FUNCTION f_MessageSet : BOOL
VAR_INPUT
  stMessage   : ST_Message;
END_VAR
VAR
  uiIndex   : INT;
  uiFound   : INT;
END_VAR

stMessage.tTime := GVL_AXIS_CTRL.gsLocalTime;

FOR uiIndex := 1 TO GVL_AXIS_CTRL.gciMaxMessage
DO
  IF (GVL_AXIS_CTRL.gatMessages[uiIndex].eType = e_MessageType.eMessageEmpty)
  THEN
    GVL_AXIS_CTRL.gatMessages[uiIndex] := stMessage;
    GVL_AXIS_CTRL.giMsgIndex := uiIndex;
    EXIT;
  END_IF
END_FOR

IF (stMessage.eType = E_MessageType.eMessageError)
THEN
  GVL_AXIS_CTRL.giErrorIndex := GVL_AXIS_CTRL.giErrorIndex + 1;
END_IF

END_FUNCTION

(* stored: Version 1.1.0.1, ProductVersion 3.1.4024.12
   POU f_MessageSet: Id {8eeea270-a0d8-4f12-86b6-de12ddb529a1}, SpecialFunc None *)
